FUNCTION_BLOCK Section2Ctrl (* Basic Function Block Type *)
  (* Standard: 61499-2 *)
  (* Version 0.0, 5/26/2018, Antti, nxtControl GmbH, Template *)
  PACKAGE Main;
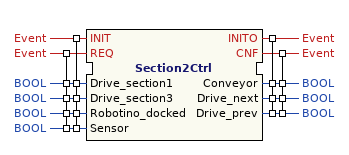
  EVENT_INPUT
    INIT WITH Drive_section1, Drive_section3, Robotino_docked, Sensor; (* Initialization Request *)
    REQ WITH Drive_section1, Drive_section3, Robotino_docked, Sensor; (* Normal Execution Request *)
  END_EVENT
  EVENT_OUTPUT
    INITO WITH Conveyor, Drive_next, Drive_prev; (* Initialization Confirm *)
    CNF WITH Conveyor, Drive_next, Drive_prev; (* Execution Confirmation *)
  END_EVENT
  VAR_INPUT
    Drive_section1 : BOOL; (* Input event qualifier *)
    Drive_section3 : BOOL;
    Robotino_docked : BOOL;
    Sensor : BOOL;
  END_VAR
  VAR_OUTPUT
    Conveyor : BOOL;
    Drive_next : BOOL; (* Output event qualifier *)
    Drive_prev : BOOL;
  END_VAR
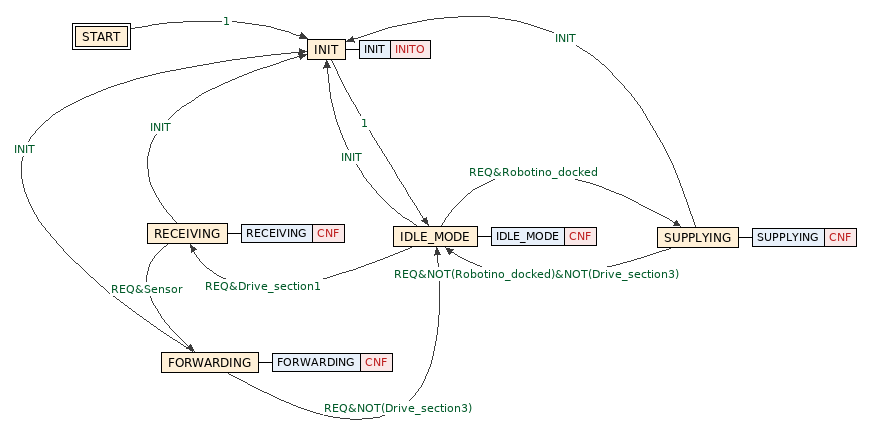
  EC_STATES
    START; (* Initial State *)
    INIT : INIT -> INITO; (* Initialization *)
    IDLE_MODE : IDLE_MODE -> CNF;
    SUPPLYING : SUPPLYING -> CNF;
    RECEIVING : RECEIVING -> CNF;
    FORWARDING : FORWARDING -> CNF;
  END_STATES
  EC_TRANSITIONS
    START TO INIT := 1;
    INIT TO IDLE_MODE := 1;
    IDLE_MODE TO SUPPLYING := REQ&Robotino_docked;
    SUPPLYING TO IDLE_MODE := REQ&NOT(Robotino_docked)&NOT(Drive_section3);
    IDLE_MODE TO RECEIVING := REQ&Drive_section1;
    RECEIVING TO FORWARDING := REQ&Sensor;
    FORWARDING TO IDLE_MODE := REQ&NOT(Drive_section3);
    IDLE_MODE TO INIT := INIT;
    SUPPLYING TO INIT := INIT;
    FORWARDING TO INIT := INIT;
    RECEIVING TO INIT := INIT;
  END_TRANSITIONS
  ALGORITHM INIT IN ST: (* Initialization algorithm *)
;
Conveyor := FALSE;
Drive_next := FALSE;
Drive_prev := FALSE;
  END_ALGORITHM
  ALGORITHM REQ IN ST: (* Normally executed algorithm *)
;
  END_ALGORITHM
  ALGORITHM IDLE_MODE IN ST:
;
Conveyor := FALSE;
Drive_next := FALSE;
Drive_prev := TRUE;
  END_ALGORITHM
  ALGORITHM SUPPLYING IN ST:
;
Conveyor := TRUE;
Drive_next := TRUE;
Drive_prev := FALSE;
  END_ALGORITHM
  ALGORITHM RECEIVING IN ST:
;
Conveyor := TRUE;
Drive_next := FALSE;
Drive_prev := TRUE;
  END_ALGORITHM
  ALGORITHM FORWARDING IN ST:
;
Conveyor := TRUE;
Drive_next := TRUE;
Drive_prev := FALSE;
  END_ALGORITHM
END_FUNCTION_BLOCK
